// TwinCAT 3 PLC project FunctionBlockPractice
// ProgramVersion: 3.1.4024.0
// libraries:
//   Tc2_Standard, * (Beckhoff Automation GmbH)
//   Tc2_System, * (Beckhoff Automation GmbH)
//   Tc2_Utilities, * (Beckhoff Automation GmbH)
//   Tc3_Module, * (Beckhoff Automation GmbH)
// project tree:
//   DUTs/ E_Event.TcDUT, ST_Event.TcDUT
//   GVLs/ GVL_Sum.TcGVL
//   / PlcTask.TcTTO
//   POUs/ AddNums.TcPOU, EventLogger.TcPOU, FB_Car.TcPOU, MAIN.TcPOU, Motor.TcPOU, UpdateTimeStampWithSystemTime.TcPOU
// real-time tasks:
//   TASK PlcTask: cycle T#10ms, priority 20, ADS port 350
//   TASK PlcTask2: cycle T#10ms, priority 22, ADS port 352
//   TASK PlcTask1: cycle T#10ms, priority 21, ADS port 351
//   TASK PlcTask3: cycle T#10ms, priority 23, ADS port 353

CONFIGURATION FunctionBlockPractice
    RESOURCE PLC ON TwinCAT3
        TASK PlcTask(INTERVAL := T#10ms, PRIORITY := 20);
        PROGRAM MAIN WITH PlcTask : MAIN;
    END_RESOURCE
END_CONFIGURATION

// ---- DUTs/E_Event.TcDUT
{attribute 'qualified_only'}
{attribute 'strict'}
TYPE E_Event :
(
	Alarm := 0,
	Message := 1,
	Warning := 2
);
END_TYPE

// ---- DUTs/ST_Event.TcDUT
TYPE ST_Event :
STRUCT
	eEventType: E_Event;
	eEventSeverity : TcEventSeverity;
	nEventIdentity : UDINT;
	sEventText : STRING(255);
	dtTimeStamp : DATE_AND_TIME;
END_STRUCT
END_TYPE

// ---- GVLs/GVL_Sum.TcGVL
{attribute 'qualified_only'}
VAR_GLOBAL
	nNumber1 : DINT;
END_VAR

// ---- POUs/MAIN.TcPOU
PROGRAM MAIN
VAR
	eEventType1 : E_Event := E_Event.Warning;
	eEventSeverity1 : TcEventSeverity := TcEventSeverity.Critical;
	nEventIdentity1 : UDINT := 32;
	sEventText1 : STRING(255) :=  'This is a danger';
	
	EventLogger1 : EventLogger;
	fbCar : FB_Car;
	fbMotor1 : Motor;
	
	nNum1 : INT;
	nNum2 : INT := 43;
	nSum : INT;
	
	nMotorValue1 : DINT;
	nMotorValue2 : DINT;
	bMotorRunning : BOOL;
	
	bFlag : BOOL := TRUE;
END_VAR

IF bFlag THEN
	EventLogger1.AddItem(eEventType:= eEventType1,eEventSeverity := eEventSeverity1,nEventIdentity := nEventIdentity1,sEventText := sEventText1 );
	GVL_Sum.nNumber1 := GVL_Sum.nNumber1 + 1;
	nMotorValue1 := fbMotor1.nMotorValue;
	fbMotor1();
	nMotorValue2 := fbMotor1.nMotorValue;
	nSum := AddNums(fbMotor1);
	
	bFlag := FALSE;
	
	fbCar.SetCarName('Tata Nexon').Start();
END_IF

END_PROGRAM

// ---- POUs/EventLogger.TcPOU
FUNCTION_BLOCK EventLogger
VAR_INPUT
	aEventBuffer : ARRAY[1..100] OF ST_Event;
END_VAR
VAR
	nEventIndex : INT := 0;
END_VAR

METHOD AddItem : BOOL
VAR_INPUT
	eEventType: E_Event;
	eEventSeverity : TcEventSeverity;
	nEventIdentity : UDINT;
	sEventText : STRING(255);
END_VAR
IF  EventBufferisFull() THEN
	nEventIndex := nEventIndex + 1;
	aEventBuffer[nEventIndex].eEventType := eEventType;
	aEventBuffer[nEventIndex].eEventSeverity := eEventSeverity;
	aEventBuffer[nEventIndex].nEventIdentity := nEventIdentity;
	aEventBuffer[nEventIndex].sEventText := sEventText;
	UpdateTimeStampWithSystemTime(stEvent := aEventBuffer[nEventIndex]);
	
	AddItem := TRUE;
ELSE
	AddItem := FALSE;
END_IF
END_METHOD

METHOD PRIVATE EventBufferisFull : BOOL
VAR_INPUT
END_VAR
IF nEventIndex > 100 THEN
	EventBufferisFull := FALSE;
ELSE
	EventBufferisFull := TRUE;
END_IF
END_METHOD

END_FUNCTION_BLOCK

// ---- POUs/UpdateTimeStampWithSystemTime.TcPOU
FUNCTION UpdateTimeStampWithSystemTime : BOOL
VAR_INPUT
	stEvent : REFERENCE TO ST_Event;
END_VAR
VAR
	fbGetSystemTime  : GETSYSTEMTIME;
	stFileTime : T_FILETIME;
END_VAR

fbGetSystemTime(timeLoDW => stFiletime.dwLowDateTime,
				 timeHiDW => stFileTime.dwHighDateTime);
stEvent.dtTimeStamp := FILETIME_TO_DT(fileTime := stFileTime);

END_FUNCTION

// ---- POUs/FB_Car.TcPOU
FUNCTION_BLOCK FB_Car
VAR_INPUT
END_VAR
VAR
	sCarName : STRING(300);
	fRunning : BOOL;
END_VAR

METHOD SetCarName : REFERENCE TO FB_Car
VAR_INPUT
	sCarName : STRING(300);
END_VAR
THIS^.sCarName := sCarName;
SetCarName REF= THIS^;
END_METHOD

METHOD Start : BOOL
VAR_INPUT
END_VAR
fRunning := TRUE;
END_METHOD

END_FUNCTION_BLOCK

// ---- POUs/Motor.TcPOU
FUNCTION_BLOCK Motor
VAR_INPUT
	nMotorNum :DINT ;
END_VAR
VAR_OUTPUT
	nMotorValue : DINT;
END_VAR
VAR
	nMotorSpin : DINT;
END_VAR

nMotorSpin := nMotorSpin + 1;

END_FUNCTION_BLOCK

// ---- POUs/AddNums.TcPOU
FUNCTION AddNums : INT
VAR_IN_OUT
	fbMotor1 :Motor;
END_VAR
VAR
	nNum1 :INT ;
	fbMotor2 :Motor;
END_VAR


IF __ISVALIDREF(fbMotor1) THEN
	//AddNums := 1/nNum1;
	
END_IF

END_FUNCTION
